// TIA Portal V17 export
// export: Created 2024-09-02T12:50:40.8160964Z, ExportSetting WithDefaults, DisplayName Totally Integrated Automation Portal, DisplayVersion V17, DisplayName TIA Portal Openness, DisplayVersion V17, DisplayName TIA Portal Version Control Interface, DisplayVersion V17, DisplayName STEP 7 Professional, DisplayVersion V17, DisplayName STEP 7 Safety, DisplayVersion V17, DisplayName WinCC Professional, DisplayVersion V17
TYPE "Aveva_Result_General_info"
// stored: IsFailsafeCompliant false
   STRUCT
      PalletID { ExternalWritable := 'False'} : String[25];   // Unique Pallet ID/Product ID
      Timestamp { ExternalWritable := 'False'} : LDT;
      iSynchro : Int;   // Synchronization word between PLC Concentrator/PLC Workstation
      iDefault : String[50];   // Default Word
      Toggle_Button_Status { ExternalWritable := 'False'} : Bool;
      Reason_Button_Status { ExternalWritable := 'False'} : String[15];
      Product_Status { ExternalWritable := 'False'} : Int;
   END_STRUCT;
END_TYPE
